(*
SPDX-FileCopyrightText: © 2026 Oleksandr Tiutyk <trofimich@gmail.com>
SPDX-License-Identifier: MIT
License: https://opensource.org/license/mit
*)

{attribute 'no_explicit_call' := 'do not call this function block directly'} 
PROGRAM ExceptionManager
VAR
	{attribute 'hide'} 
	_ClassName : STRING := __POUNAME();

	_Exception : IException;
	_SystemException : SystemException;
END_VAR

{attribute 'monitoring' := 'call'}
PROPERTY ClassName : REFERENCE TO STRING
GET
ClassName REF= _ClassName;
END_GET
END_PROPERTY

(*!
<summary>Drops the borrowed framework payload before DynamicMemoryManager deletes registered objects.</summary>
<description>
Does not delete exceptions or reset the shared SystemException.
</description>
*)

METHOD Cleanup
_Exception := 0;
END_METHOD

(*!
<summary>Returns the framework payload or the shared SystemException configured for this catch.</summary>
<description>
The result is borrowed; the shared system instance changes on the next system catch.
Clone a static result before callbacks that may handle another system error.
A SystemException propagated by Throw is a dynamic framework payload retaining its original metadata.
A native code already lost by the runtime cannot be reconstructed here.
</description>
*)

METHOD GetLastException : IException
VAR_INPUT 
	exceptionCode : __SYSTEM.ExceptionCode;
	catchPointNamespaceName : STRING;
	catchPointPOUName : STRING;
	catchPointPosition : STRING;
END_VAR
// 3902013441 is a workaround for bug in 3.1.4026.19
IF (exceptionCode = __SYSTEM.ExceptionCode.RTSEXCPT_USER_EXCEPTION_BASE OR_ELSE exceptionCode = 3902013441) AND_THEN _Exception <> 0 THEN
	GetLastException := _Exception;
ELSE
	_SystemException.Configure(exceptionCode, catchPointNamespaceName, catchPointPOUName, catchPointPosition);
	GetLastException := _SystemException;
END_IF
END_METHOD

{attribute 'monitoring' := 'call'}
PROPERTY NamespaceName : REFERENCE TO STRING
GET
NamespaceName REF= CurrentNamespace.Name;
END_GET
END_PROPERTY

(*!
<summary>Propagates the current exception as a framework payload, wrapping native errors in SystemException.</summary>
<description>
Pass the current catch code and its location, or the exception already obtained for that catch.
A supplied exception takes precedence over the code and preserves its original catch point and timestamps.
Before callbacks that can handle another error, clone a borrowed static SystemException and retain that clone.
Static payloads are cloned on propagation; dynamic payloads retain identity until automatic cleanup.
The next raw catch code identifies framework transport, not the original native error.
A latched allocation failure is raised before any allocation and is never wrapped here.
</description>
*)

METHOD ReThrowLastException
VAR_INPUT
	exceptionCode : __SYSTEM.ExceptionCode;
	exception : IException := 0;
	catchPointNamespaceName : STRING := '';
	catchPointPOUName : STRING := '';
	catchPointPosition : STRING := '';
END_VAR
VAR
	currentException : IException;
END_VAR
DynamicMemoryManager.RaiseIfAllocationFailed();

currentException := exception;
IF currentException = 0 THEN
	currentException := GetLastException(exceptionCode, catchPointNamespaceName, catchPointPOUName, catchPointPosition);
END_IF

Throw(currentException);
END_METHOD

(*!
<summary>Null is a no-op. Dynamic exceptions are borrowed; static exceptions are cloned.</summary>
<description>
The clone must implement IException and have a lifetime covering all handlers until cleanup.
Framework implementations register dynamic clones with DynamicMemoryManager.
SystemException uses the same transport and retains its captured native code and timestamps.
A latched allocation failure is raised before cloning.
</description>
*)

METHOD Throw
VAR_INPUT CONSTANT
	exception : IException;
END_VAR
IF exception = 0 THEN
	RETURN;
END_IF

DynamicMemoryManager.RaiseIfAllocationFailed();

//LogManager.TryLogException(exception, "Exception", "Exception.Throw", WideStrings.Concat255(STRING_TO_WSTRING(exception.ClassName), ".Throw"));

IF exception.IsDynamicInstance THEN
	_Exception := exception;
ELSE
	__QUERYINTERFACE(exception.Clone(), _Exception);
END_IF

Tc2_System.F_RaiseException(__SYSTEM.ExceptionCode.RTSEXCPT_USER_EXCEPTION_BASE);
END_METHOD

END_PROGRAM

(* stored: Version 1.1.0.1
   POU ExceptionManager: Id {a83d007f-42e6-48cd-9a14-7b9a497b4ddf}, SpecialFunc None
   Property ClassName: Id {48fade2e-63bd-4687-b635-a26e3a0e44d2}
   Get Get: Id {f78e5eeb-7174-4e7e-8bf4-5241f5dd7503}
   Method Cleanup: Id {9439ecc4-f37f-44e7-803e-1ee8d39cff59}
   Method GetLastException: Id {e2be0c6d-d285-4e57-9453-ace2efe79ed7}
   Property NamespaceName: Id {dda72a28-bb72-497e-8f27-b037ac7ca94f}
   Get Get: Id {db04ba72-0d5b-4d3e-bca2-301f74e7a26c}
   Method ReThrowLastException: Id {7ea9eaf2-899d-4c20-8cad-4853167d967f}
   Method Throw: Id {75adab3e-0cb1-497b-afc4-6a0aa273ac06} *)
